// TIA Portal project "RFID_0" (V20)

(* hardware
DEVICE "S7-1500/ET200MP-Station_1"  S7-1500 station
   slot 0: "Profilschiene_0"  Rack  6ES7 590-1***0-0AA0
   slot 1: "PLC_1"  CPU 1515-2 PN  6ES7 515-2AM02-0AB0  V2.9
      slot 3: "CPU-Display_1"  6ES7591-1BA00-0AA0
      slot 32768: "PROFINET-Schnittstelle_1"  X1
         slot 32769: "Port_1"  X1 P1
         slot 32770: "Port_2"  X1 P2
      slot 33024: "PROFINET-Schnittstelle_2"  X2
         slot 33025: "Port_1"  X2 P1
      slot 34817: "Virtual CP interface port_1"  Virtual CP interface port  Virtual CP interface port
   slot 2: "AI 8xU/I/R/RTD BA_1"  AI 8xU/I/R/RTD BA  6ES7 531-7QF00-0AB0  V1.0
   slot 3: "AI 8xU/I/R/RTD BA_2"  AI 8xU/I/R/RTD BA  6ES7 531-7QF00-0AB0  V1.0
   slot 4: "AI 8xU/I/R/RTD BA_3"  AI 8xU/I/R/RTD BA  6ES7 531-7QF00-0AB0  V1.0
   slot 5: "AQ 8xU/I HS_1"  AQ 8xU/I HS  6ES7 532-5HF00-0AB0  V2.2
   slot 6: "AQ 8xU/I HS_2"  AQ 8xU/I HS  6ES7 532-5HF00-0AB0  V2.2
   slot 7: "AQ 8xU/I HS_3"  AQ 8xU/I HS  6ES7 532-5HF00-0AB0  V2.2
*)

// ===== PLC "PLC_1"  CPU 1515-2 PN =====

VAR_GLOBAL   // PLC tag table "Eingaenge"
   "1B1" AT %I0.0 : Bool;   // Sensor (Ein)
   "1B3" AT %I0.1 : Bool;   // Sensor (Aus)
   "FACTORY I/O (Running)" AT %I0.7 : Bool;
   "1B2" AT %ID30 : DInt;   // Visionsensor
   "Status_1" AT %ID34 : DInt;   // RFID_1 Status
   "Read_1" AT %ID38 : DInt;   // RFID_1 Read Data
   "ComID_1" AT %ID42 : DInt;   // RFID_1 Command ID
   "Status_2" AT %ID50 : DInt;   // RFID_2 Status
   "Read_2" AT %ID54 : DInt;   // RFID_2 Read Data
   "ComID_2" AT %ID58 : DInt;   // RFID_2 Command ID
   "Status_3" AT %ID66 : DInt;   // RFID_3 Status
   "Read_3" AT %ID70 : DInt;   // RFID_3 Read Data
   "ComID_3" AT %ID74 : DInt;   // RFID_3 Command ID
END_VAR

VAR_GLOBAL   // PLC tag table "Ausgaenge"
   "1M1" AT %Q0.0 : Bool;   // Band
   "ExecCom_1" AT %Q0.2 : Bool;   // RFID_1 Execute Command
   "ExecCom_2" AT %Q0.3 : Bool;   // RFID_2 Execute Command
   "ExecCom_3" AT %Q0.4 : Bool;   // RFID_3 Execute Command
   "Com_1" AT %QD34 : DInt;   // RFID_1 Command
   "Write_1" AT %QD38 : DInt;   // RFID_1 Write Data
   "MemInd_1" AT %QD42 : DInt;   // RFID_1 Memory Index
   "Com_2" AT %QD50 : DInt;   // RFID_2 Command
   "Write_2" AT %QD54 : DInt;   // RFID_2 Write Data
   "MemInd_2" AT %QD58 : DInt;   // RFID_2 Memory Index
   "Com_3" AT %QD66 : DInt;   // RFID_3 Command
   "Write_3" AT %QD70 : DInt;   // RFID_3 Write Data
   "MemInd_3" AT %QD74 : DInt;   // RFID_3 Memory Index
END_VAR

TYPE "typEingaenge"
   STRUCT
      "1B1" : Bool;
      "1B2" : DInt;
      "1B3" : Bool;
   END_STRUCT;
END_TYPE

TYPE "typAusgaenge"
   STRUCT
      "1M1" : Bool;
   END_STRUCT;
END_TYPE

TYPE "typRFID"
   STRUCT
      In : Struct
         Status : DInt;
         ReadData : DInt;
         CommandID : DInt;
      END_STRUCT;
      Out : Struct
         ExecuteCommand : Bool;
         Command : DInt;
         WriteData : DInt;
         MemoryIndex : DInt;
      END_STRUCT;
   END_STRUCT;
END_TYPE

TYPE "typRFID_Daten"
   STRUCT
      ID : DInt;
      Daten : Array[0..2] of DInt;
   END_STRUCT;
END_TYPE

DATA_BLOCK "IDB_Anlage_ein"   // DB1
{ S7_Optimized_Access := 'TRUE' }
VERSION : 0.1
// stored: InstanceOfName Anlage_ein
"Anlage_ein"
BEGIN
END_DATA_BLOCK

DATA_BLOCK "Bandsteuerung_DB"   // DB10
{ S7_Optimized_Access := 'TRUE' }
VERSION : 0.1
// stored: InstanceOfName Bandsteuerung
"Bandsteuerung"
BEGIN
END_DATA_BLOCK

DATA_BLOCK "Read_RFID_DB"   // DB20
{ S7_Optimized_Access := 'TRUE' }
VERSION : 0.1
// stored: InstanceOfName Read_RFID
"Read_RFID"
BEGIN
END_DATA_BLOCK

DATA_BLOCK "Write_RFID_DB"   // DB21
{ S7_Optimized_Access := 'TRUE' }
VERSION : 0.1
// stored: InstanceOfName Write_RFID
"Write_RFID"
BEGIN
END_DATA_BLOCK

DATA_BLOCK "Read_RFID_DB2"   // DB22
{ S7_Optimized_Access := 'TRUE' }
VERSION : 0.1
// stored: InstanceOfName Read_RFID
"Read_RFID"
BEGIN
END_DATA_BLOCK

DATA_BLOCK "HMI"   // DB100
{ S7_Optimized_Access := 'TRUE' }
VERSION : 0.1
   VAR
      Eingaenge : "typEingaenge";
      Ausgaenge : "typAusgaenge";
      RFID_Geraet : Array[0..2] of "typRFID";
      Anlagedaten : Struct
         Bauteil : DInt;
         CurRFID : DInt;
      END_STRUCT;
   END_VAR
BEGIN
END_DATA_BLOCK

DATA_BLOCK "DB_Register"   // DB999
{ S7_Optimized_Access := 'TRUE' }
VERSION : 0.1
   VAR
      Register : Array[0..3] of "typRFID_Daten";
   END_VAR
BEGIN
END_DATA_BLOCK

FUNCTION_BLOCK "Anlage_ein"   // FB1, FBD
{ S7_Optimized_Access := 'TRUE' }
VERSION : 0.1
   VAR
      MI_RTRIG_1B1 : R_TRIG;
      MI_FTRIG_1B1 : F_TRIG;
      MI_RTRIG_1B2 : R_TRIG;
      MI_FTRIG_1B2 : F_TRIG;
      MI_RTRIG_1B3 : R_TRIG;
      MI_FTRIG_1B3 : F_TRIG;
   END_VAR
BEGIN

REGION Network 1 (SCL)
   // Bits
   "HMI".Eingaenge."1B1" := "1B1";
   "HMI".Eingaenge."1B3" := "1B3";

   // Word
   "HMI".Eingaenge."1B2" := "1B2";

   "HMI".RFID_Geraet[0].In.Status := "Status_1";
   "HMI".RFID_Geraet[0].In.ReadData := "Read_1";
   "HMI".RFID_Geraet[0].In.CommandID := "ComID_1";

   "HMI".RFID_Geraet[1].In.Status := "Status_2";
   "HMI".RFID_Geraet[1].In.ReadData := "Read_2";
   "HMI".RFID_Geraet[1].In.CommandID := "ComID_2";

   "HMI".RFID_Geraet[2].In.Status := "Status_3";
   "HMI".RFID_Geraet[2].In.ReadData := "Read_3";
   "HMI".RFID_Geraet[2].In.CommandID := "ComID_3";
END_REGION

REGION Network 2 (SCL): Flanken
   #MI_RTRIG_1B1(CLK := "1B1");
   #MI_FTRIG_1B1(CLK := "1B1");
   #MI_RTRIG_1B2(CLK := "1B2" <> 0);
   #MI_FTRIG_1B2(CLK := "1B2" <> 0);
   #MI_RTRIG_1B3(CLK := "1B3");
   #MI_FTRIG_1B3(CLK := "1B3");
END_REGION
END_FUNCTION_BLOCK

FUNCTION_BLOCK "Bandsteuerung"   // FB10, FBD
{ S7_Optimized_Access := 'TRUE' }
VERSION : 0.1
   VAR_INPUT
      Band_weiter : Bool;
      RTRIG_1B1 : Bool;
   END_VAR
   VAR_IN_OUT
      Band : Bool;
   END_VAR
   VAR
      RTRIG_FactoryRunning : R_TRIG;
   END_VAR
BEGIN

REGION Network 1: Flanken
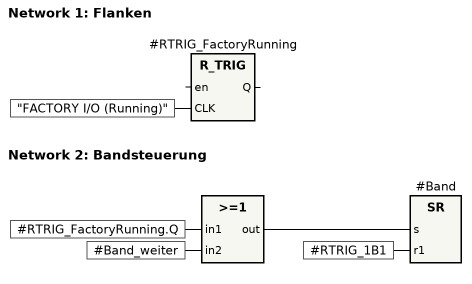
   #RTRIG_FactoryRunning(CLK := "FACTORY I/O (Running)");   // R_TRIG
END_REGION

REGION Network 2: Bandsteuerung
   IF #RTRIG_FactoryRunning.Q OR #Band_weiter THEN
       #Band := TRUE;   // SR flip-flop
   END_IF;
   IF #RTRIG_1B1 THEN #Band := FALSE; END_IF;
END_REGION
END_FUNCTION_BLOCK

FUNCTION_BLOCK "Read_RFID"   // FB20, FBD
{ S7_Optimized_Access := 'TRUE' }
VERSION : 0.1
   VAR_INPUT
      RTRIG_Trigger : Bool;
      CommandType : DInt;   // Die Art des Kommandos (siehe Factory Handbuch).
      ComID : DInt;   // Die neue Kommdo ID vom RFID Reader.
      Read : DInt;   // Die Daten aus dem RFID Reader.
      Status : DInt;   // Der Status, der vom ausgeführten Kommando aus dem Reader-Anschluss zurückkommt.
   END_VAR
   VAR_OUTPUT
      Band_weiter : Bool;
      ComType : DInt;   // Reader-Anschluss, wo das Kommando gesetzt wird.
   END_VAR
   VAR_IN_OUT
      ExecCom : Bool;   // Reader-Anschluss bei dem das Kommando ausgeführt werden soll.
      MemInd : DInt;
   END_VAR
   VAR
      Reader_CommandID : DInt;   // Letzes hochgezähltes Kommando Inkrement.
      TP_RFID : TP_TIME;
      FTRIG_TP : F_TRIG;
   END_VAR
BEGIN

REGION Network 1: Timer
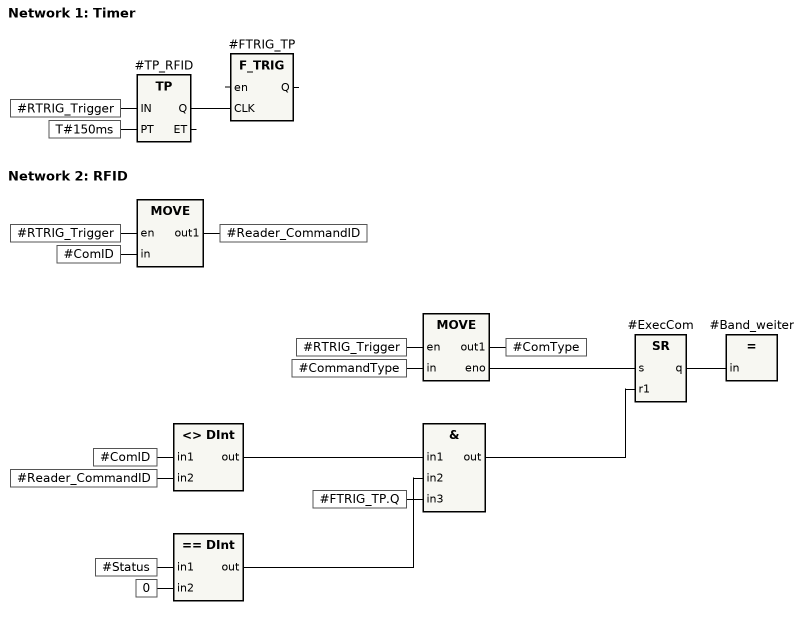
   #TP_RFID(IN := #RTRIG_Trigger, PT := T#150ms);   // TP
   #FTRIG_TP(CLK := #TP_RFID.Q);   // F_TRIG
END_REGION

REGION Network 2: RFID
   // ID auslesen
   // mit erfolgreichem Kommando das ausgeführte Kommando zurücksetzen.
   IF #RTRIG_Trigger THEN
       #Reader_CommandID := #ComID;
       #ComType := #CommandType;
       #ExecCom := TRUE;   // SR flip-flop
   END_IF;
   IF (#ComID <> #Reader_CommandID) AND (#Status = 0) AND #FTRIG_TP.Q THEN #ExecCom := FALSE; END_IF;
   #Band_weiter := #ExecCom;
END_REGION

REGION Network 3 (SCL)
   IF #ExecCom THEN
       IF #CommandType = 1 THEN
           "DB_Register".Register[0].ID := #Read;
       ELSIF #CommandType = 2 THEN
           "DB_Register".Register[2].Daten[#MemInd] := #Read;
       END_IF;
   END_IF;
END_REGION
END_FUNCTION_BLOCK

FUNCTION_BLOCK "Write_RFID"   // FB21, FBD
{ S7_Optimized_Access := 'TRUE' }
VERSION : 0.1
   VAR_INPUT
      VisionSensor : DInt;
      RTRIG_Trigger : Bool;
      ComID : DInt;
      Status : DInt;
   END_VAR
   VAR_OUTPUT
      ComType : DInt;
      Write : DInt;
   END_VAR
   VAR_IN_OUT
      ExecCom : Bool;
      MemInd : DInt;
   END_VAR
   VAR
      Reader_CommandID : DInt;
   END_VAR
BEGIN

REGION Network 1
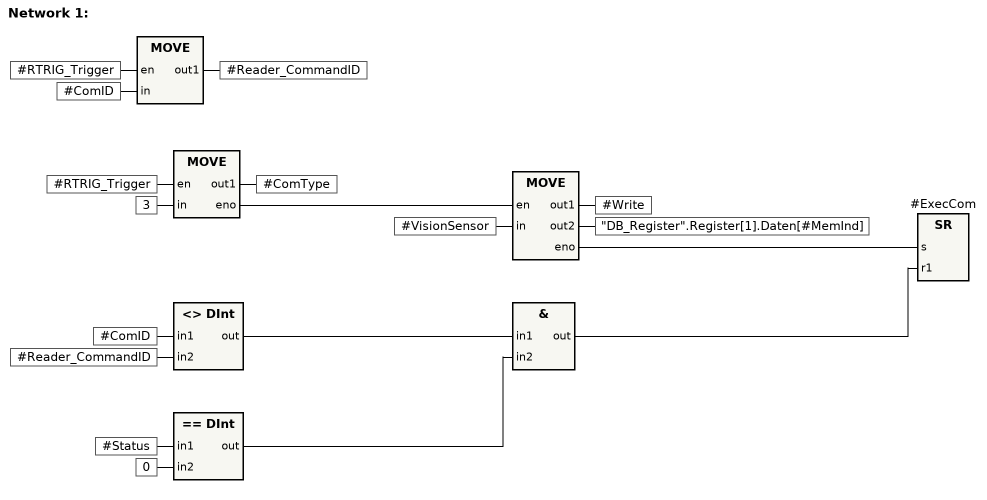
   IF #RTRIG_Trigger THEN
       #Reader_CommandID := #ComID;
       #ComType := 3;
       #Write := #VisionSensor;
       "DB_Register".Register[1].Daten[#MemInd] := #VisionSensor;
       #ExecCom := TRUE;   // SR flip-flop
   END_IF;
   IF (#ComID <> #Reader_CommandID) AND (#Status = 0) THEN #ExecCom := FALSE; END_IF;
END_REGION
END_FUNCTION_BLOCK

FUNCTION "Anlage_aus" : Void   // FC1, FBD
{ S7_Optimized_Access := 'TRUE' }
VERSION : 0.1
BEGIN

REGION Network 1 (SCL): Band
   // Bits
   "1M1" := "HMI".Ausgaenge."1M1";

   "ExecCom_1" := "HMI".RFID_Geraet[0].Out.ExecuteCommand;
   "ExecCom_2" := "HMI".RFID_Geraet[1].Out.ExecuteCommand;
   "ExecCom_3" := "HMI".RFID_Geraet[2].Out.ExecuteCommand;


   // Word
   "Com_1" := "HMI".RFID_Geraet[0].Out.Command;
   "Write_1" := "HMI".RFID_Geraet[0].Out.WriteData;
   "MemInd_1" := "HMI".RFID_Geraet[0].Out.MemoryIndex;

   "Com_2" :="HMI".RFID_Geraet[1].Out.Command;
   "Write_2" := "HMI".RFID_Geraet[1].Out.WriteData;
   "MemInd_2" := "HMI".RFID_Geraet[1].Out.MemoryIndex;

   "Com_3" :="HMI".RFID_Geraet[2].Out.Command;
   "Write_3" :="HMI".RFID_Geraet[2].Out.WriteData;
   "MemInd_3" := "HMI".RFID_Geraet[2].Out.MemoryIndex;
END_REGION
END_FUNCTION

FUNCTION "Schieberegister" : Void   // FC2, FBD
{ S7_Optimized_Access := 'TRUE' }
VERSION : 0.1
   VAR_INPUT
      FTRIG_Trigger : Bool;
      Startindex : DInt;
      Laenge : DInt;
   END_VAR
   VAR_IN_OUT
      Register : Array[*] of "typRFID_Daten";
   END_VAR
   VAR_TEMP
      i : DInt;
   END_VAR
BEGIN

REGION Network 1 (SCL): Schieberegister
   // Schieben, wenn Palette an Sensor vorbei ist.
   IF #FTRIG_Trigger THEN
       FOR #i := 3 TO 1 BY -1 DO
           #Register[#i] := #Register[#i - 1];
       END_FOR;

       #Register[0].ID := 0;
   END_IF;
END_REGION
END_FUNCTION

ORGANIZATION_BLOCK "Main"   // OB1, FBD, ProgramCycle
TITLE = "Main Program Sweep (Cycle)"
{ S7_Optimized_Access := 'TRUE' }
VERSION : 0.1
   VAR_INPUT
      Initial_Call : Bool;   // Initial call of this OB
      Remanence : Bool;   // =True, if remanent data are available
   END_VAR
   VAR_TEMP
      Band_weiter1 : Bool;
      Band_weiter2 : Bool;
   END_VAR
BEGIN

REGION Network 1
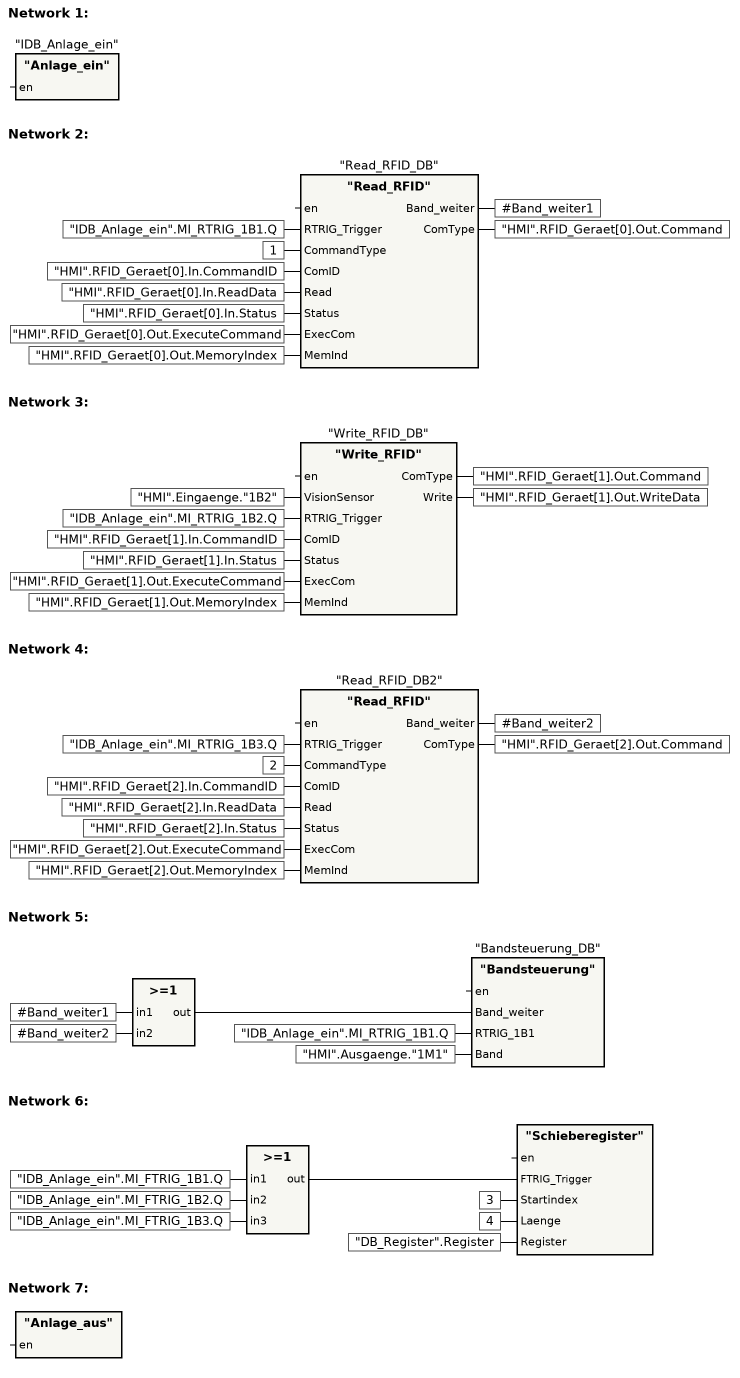
   "IDB_Anlage_ein"();   // "Anlage_ein"
END_REGION

REGION Network 2
   "Read_RFID_DB"(RTRIG_Trigger := "IDB_Anlage_ein".MI_RTRIG_1B1.Q,   // "Read_RFID"
                  CommandType := 1,
                  ComID := "HMI".RFID_Geraet[0].In.CommandID,
                  Read := "HMI".RFID_Geraet[0].In.ReadData,
                  Status := "HMI".RFID_Geraet[0].In.Status,
                  ExecCom := "HMI".RFID_Geraet[0].Out.ExecuteCommand,
                  MemInd := "HMI".RFID_Geraet[0].Out.MemoryIndex,
                  Band_weiter => #Band_weiter1,
                  ComType => "HMI".RFID_Geraet[0].Out.Command);
END_REGION

REGION Network 3
   "Write_RFID_DB"(VisionSensor := "HMI".Eingaenge."1B2",   // "Write_RFID"
                   RTRIG_Trigger := "IDB_Anlage_ein".MI_RTRIG_1B2.Q,
                   ComID := "HMI".RFID_Geraet[1].In.CommandID,
                   Status := "HMI".RFID_Geraet[1].In.Status,
                   ExecCom := "HMI".RFID_Geraet[1].Out.ExecuteCommand,
                   MemInd := "HMI".RFID_Geraet[1].Out.MemoryIndex,
                   ComType => "HMI".RFID_Geraet[1].Out.Command,
                   Write => "HMI".RFID_Geraet[1].Out.WriteData);
END_REGION

REGION Network 4
   "Read_RFID_DB2"(RTRIG_Trigger := "IDB_Anlage_ein".MI_RTRIG_1B3.Q,   // "Read_RFID"
                   CommandType := 2,
                   ComID := "HMI".RFID_Geraet[2].In.CommandID,
                   Read := "HMI".RFID_Geraet[2].In.ReadData,
                   Status := "HMI".RFID_Geraet[2].In.Status,
                   ExecCom := "HMI".RFID_Geraet[2].Out.ExecuteCommand,
                   MemInd := "HMI".RFID_Geraet[2].Out.MemoryIndex,
                   Band_weiter => #Band_weiter2,
                   ComType => "HMI".RFID_Geraet[2].Out.Command);
END_REGION

REGION Network 5
   "Bandsteuerung_DB"(Band_weiter := #Band_weiter1 OR #Band_weiter2,   // "Bandsteuerung"
                      RTRIG_1B1 := "IDB_Anlage_ein".MI_RTRIG_1B1.Q,
                      Band := "HMI".Ausgaenge."1M1");
END_REGION

REGION Network 6
   "Schieberegister"(FTRIG_Trigger := "IDB_Anlage_ein".MI_FTRIG_1B1.Q OR "IDB_Anlage_ein".MI_FTRIG_1B2.Q OR "IDB_Anlage_ein".MI_FTRIG_1B3.Q,
                     Startindex := 3,
                     Laenge := 4,
                     Register := "DB_Register".Register);
END_REGION

REGION Network 7
   "Anlage_aus"();
END_REGION
END_ORGANIZATION_BLOCK